{attribute 'qualified_only'}
VAR_GLOBAL
	control : RemoteControl;
	feedback : RemoteFeedback;
END_VAR

(* stored: Version 1.1.0.1, ProductVersion 3.1.4020.12
   GVL REMOTE: Id {c58f8bc8-d042-42ac-b06f-9f009d98a2aa} *)
